(* CoDeSys 2.3 export: CILINDRO_SIMPLE.EXP *)

(* Data type *)
TYPE Cilindro_Simple :
STRUCT
	Valvula                       : EV_Simple;
	Sensor_Avance       : Sensor_Magnetico;
	Sensor_Retroceso : Sensor_Magnetico;
END_STRUCT
END_TYPE
